PROGRAM prgComEffIO
VAR
	fbCom		: FB_MqttCommunicator_v3;

END_VAR

fbCom(
	bConnect:= TRUE, 
	strAuthkey := 'DEV01673741737',
	sUserName:= '860e8e24-eac9-4d3f-a049-218c33986af5' , 		
	sUserPassword:= '7ff1f7e7-8e89-474f-a2a7-76bbe44eafe4',
	eSavePositionCertificate:= eSavePositionOnPLC.ePostionC, 
	bConnected=> , 
	bError=> , 
	hrErrorCode=> , 
	eConnectionState=> , 
	eErrorMessage_Out=> );

END_PROGRAM

(* stored: Version 1.1.0.1, ProductVersion 3.1.4024.12
   POU prgComEffIO: Id {7c131c8e-9f5f-4e63-8194-730ced908ef8}, SpecialFunc None *)
